FUNCTION_BLOCK FB_ErrorSource EXTENDS FB_HasInstanceName IMPLEMENTS I_HasErrorSourcing
VAR
	_errorSource	: ST_ErrorSource := (InstanceName := GetInstanceName());
END_VAR

PROPERTY ErrorSource : REFERENCE TO ST_ErrorSource
GET
ErrorSource := _errorSource;
END_GET
END_PROPERTY

END_FUNCTION_BLOCK

(* stored: Version 1.1.0.1, ProductVersion 3.1.4024.13
   POU FB_ErrorSource: Id {39c13ed9-6860-004f-28d1-bfe8a964ba5b}, SpecialFunc None
   Property ErrorSource: Id {15c87816-e531-04de-26f6-1439ba97e2e1}
   Get Get: Id {02786464-5879-0c4a-39ea-a502d632abf5} *)
